// SIMATIC S7-200 project (STEP 7-Micro/WIN), CPU 224 REL 02.01

ORGANIZATION_BLOCK MAIN:OB1
TITLE=程序注释
BEGIN
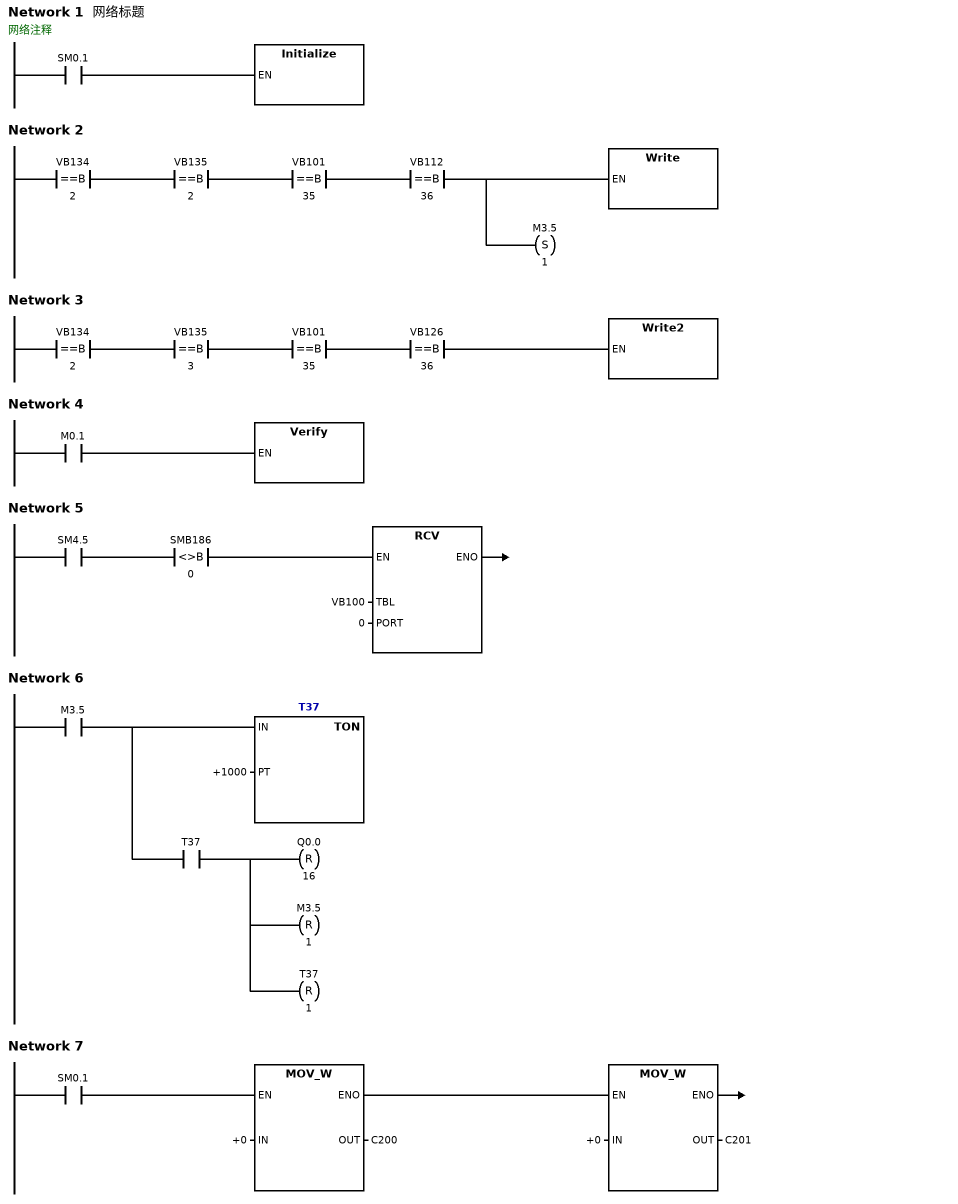
Network 1 // 网络标题
// 网络注释
LD     SM0.1
CALL   Initialize:SBR3
Network 2
LDB=   VB134, 2
AB=    VB135, 2
AB=    VB101, 35
AB=    VB112, 36
CALL   Write:SBR1
S      M3.5, 1
Network 3
LDB=   VB134, 2
AB=    VB135, 3
AB=    VB101, 35
AB=    VB126, 36
CALL   Write2:SBR6
Network 4
LD     M0.1
CALL   Verify:SBR2
Network 5
LD     SM4.5
AB<>   SMB186, 0
RCV    VB100, 0
Network 6
LD     M3.5
TON    T37, +1000
A      T37
R      Q0.0, 16
R      M3.5, 1
R      T37, 1
Network 7
LD     SM0.1
MOVW   +0, C200
AENO
MOVW   +0, C201
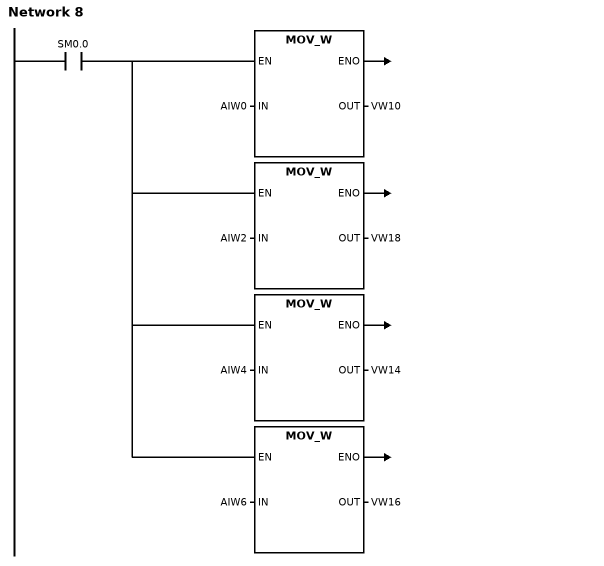
Network 8
LD     SM0.0
MOVW   AIW0, VW10
MOVW   AIW2, VW18
MOVW   AIW4, VW14
MOVW   AIW6, VW16
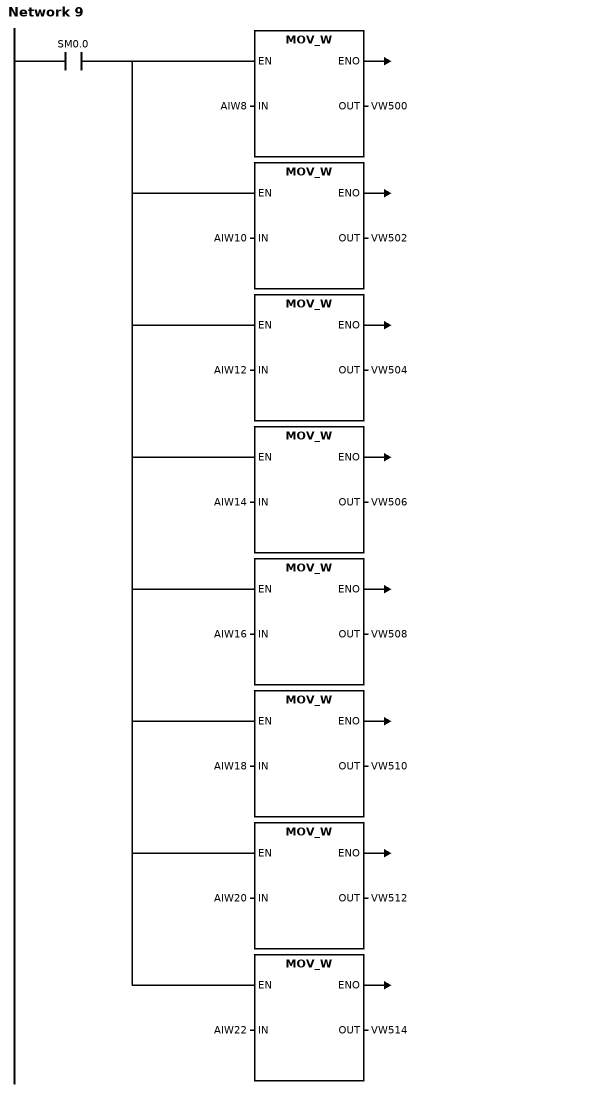
Network 9
LD     SM0.0
MOVW   AIW8, VW500
MOVW   AIW10, VW502
MOVW   AIW12, VW504
MOVW   AIW14, VW506
MOVW   AIW16, VW508
MOVW   AIW18, VW510
MOVW   AIW20, VW512
MOVW   AIW22, VW514
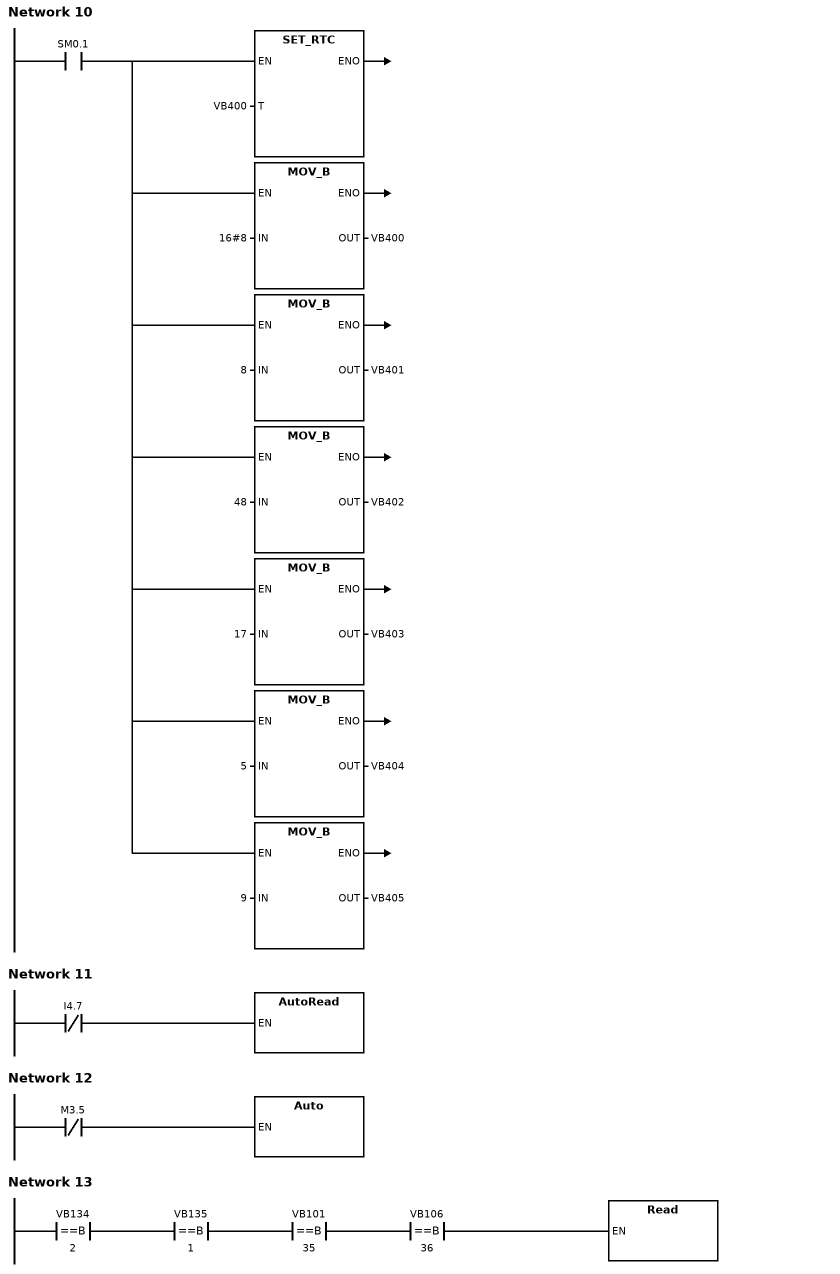
Network 10
LD     SM0.1
TODW   VB400
MOVB   16#8, VB400
MOVB   8, VB401
MOVB   48, VB402
MOVB   17, VB403
MOVB   5, VB404
MOVB   9, VB405
Network 11
LDN    I4.7
CALL   AutoRead:SBR5
Network 12
LDN    M3.5
CALL   Auto:SBR4
Network 13
LDB=   VB134, 2
AB=    VB135, 1
AB=    VB101, 35
AB=    VB106, 36
CALL   Read:SBR0
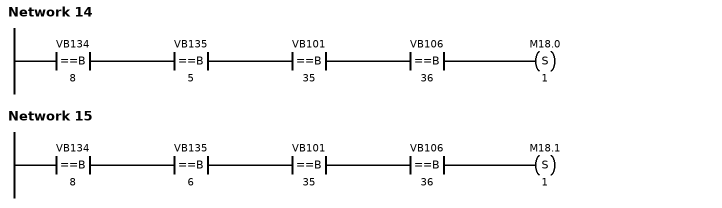
Network 14
LDB=   VB134, 8
AB=    VB135, 5
AB=    VB101, 35
AB=    VB106, 36
S      M18.0, 1
Network 15
LDB=   VB134, 8
AB=    VB135, 6
AB=    VB101, 35
AB=    VB106, 36
S      M18.1, 1
END_ORGANIZATION_BLOCK

SUBROUTINE_BLOCK Read:SBR0
TITLE=子程序注释
BEGIN
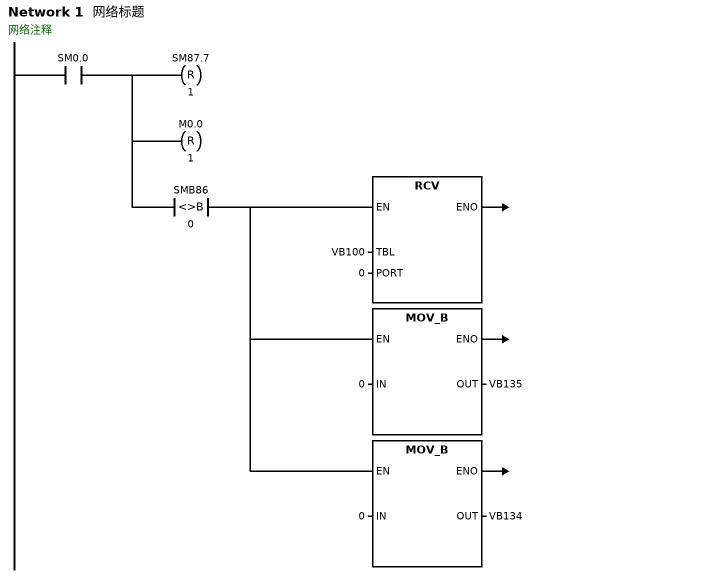
Network 1 // 网络标题
// 网络注释
LD     SM0.0
R      SM87.7, 1
R      M0.0, 1
AB<>   SMB86, 0
RCV    VB100, 0
MOVB   0, VB135
MOVB   0, VB134
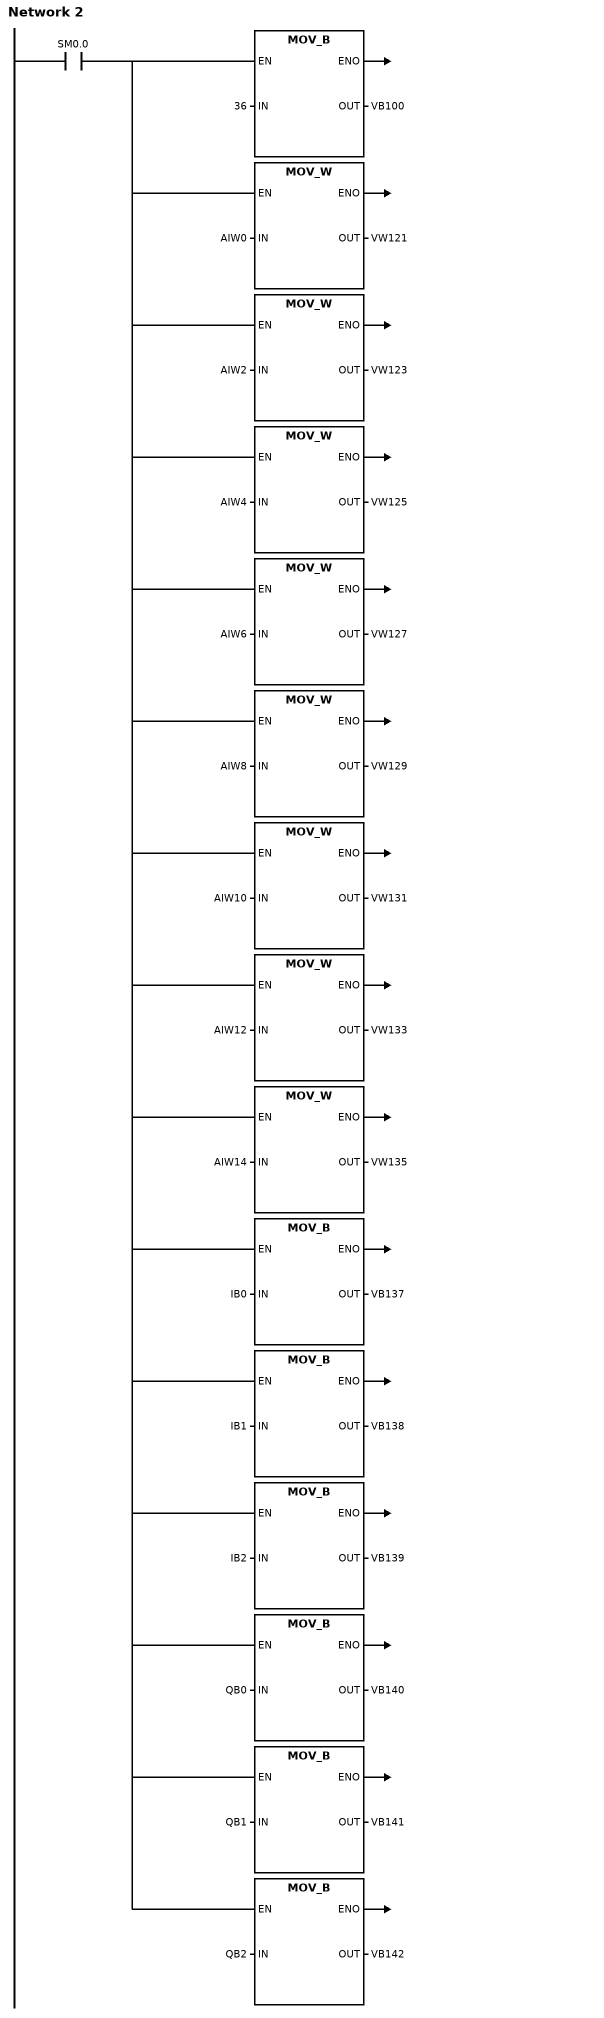
Network 2
LD     SM0.0
MOVB   36, VB100
MOVW   AIW0, VW121
MOVW   AIW2, VW123
MOVW   AIW4, VW125
MOVW   AIW6, VW127
MOVW   AIW8, VW129
MOVW   AIW10, VW131
MOVW   AIW12, VW133
MOVW   AIW14, VW135
MOVB   IB0, VB137
MOVB   IB1, VB138
MOVB   IB2, VB139
MOVB   QB0, VB140
MOVB   QB1, VB141
MOVB   QB2, VB142
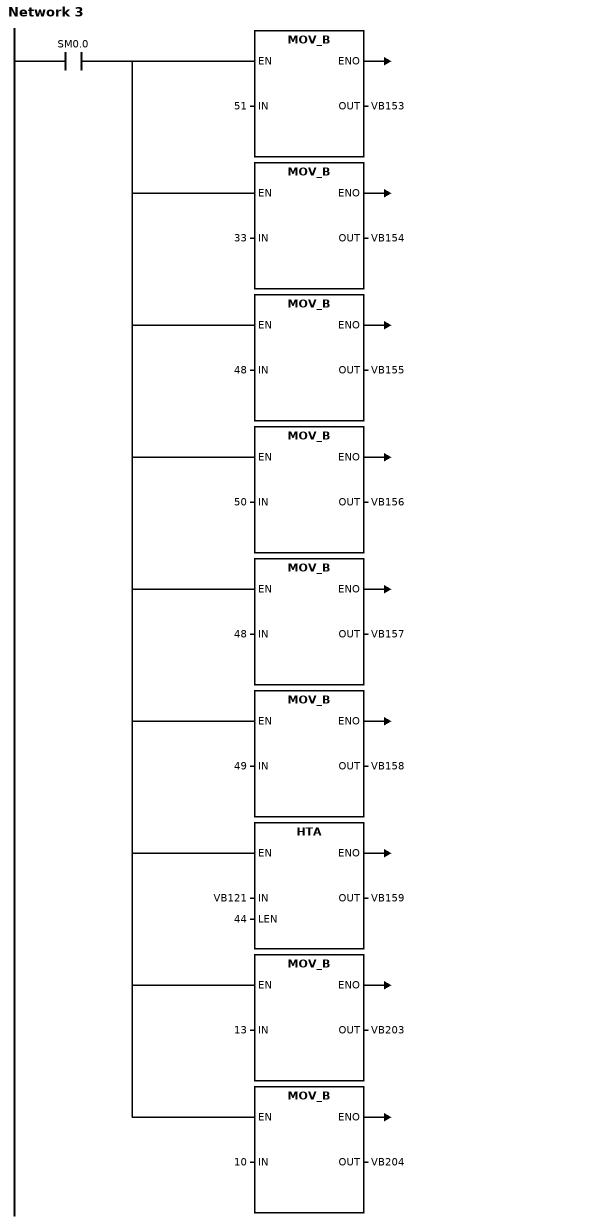
Network 3
LD     SM0.0
MOVB   51, VB153
MOVB   33, VB154
MOVB   48, VB155
MOVB   50, VB156
MOVB   48, VB157
MOVB   49, VB158
HTA    VB121, VB159, 44
MOVB   13, VB203
MOVB   10, VB204
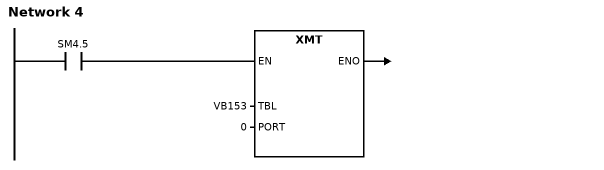
Network 4
LD     SM4.5
XMT    VB153, 0
END_SUBROUTINE_BLOCK

SUBROUTINE_BLOCK Write:SBR1
TITLE=
BEGIN
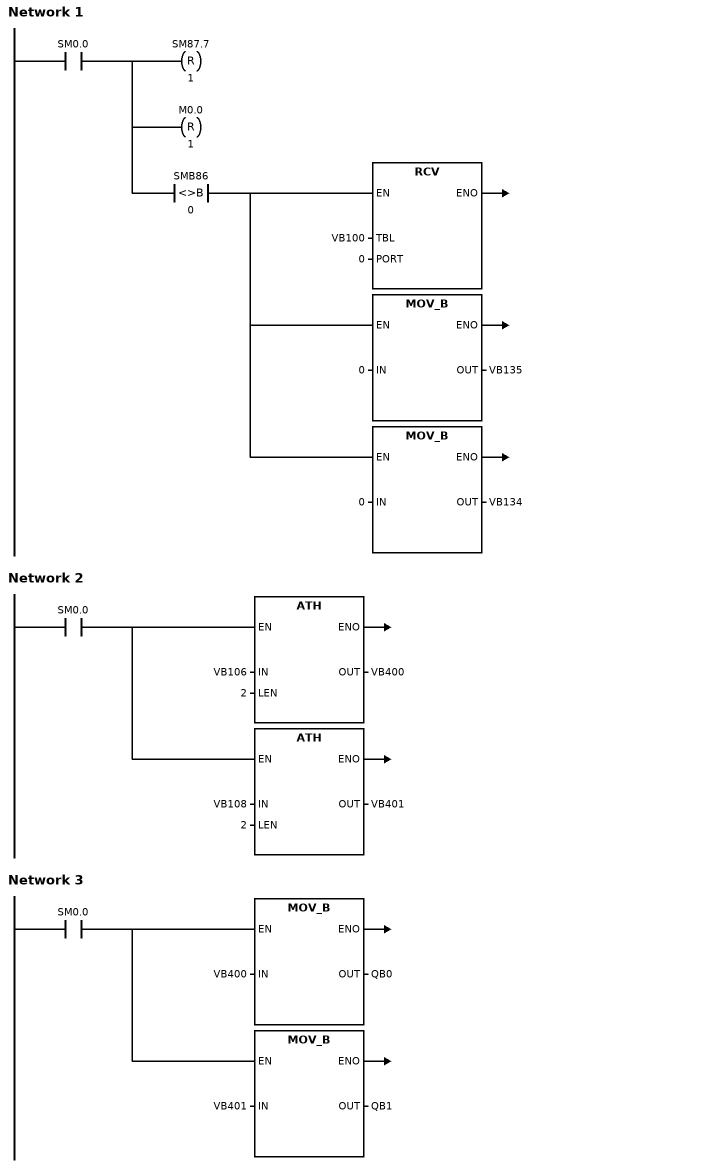
Network 1
LD     SM0.0
R      SM87.7, 1
R      M0.0, 1
AB<>   SMB86, 0
RCV    VB100, 0
MOVB   0, VB135
MOVB   0, VB134
Network 2
LD     SM0.0
ATH    VB106, VB400, 2
ATH    VB108, VB401, 2
Network 3
LD     SM0.0
MOVB   VB400, QB0
MOVB   VB401, QB1
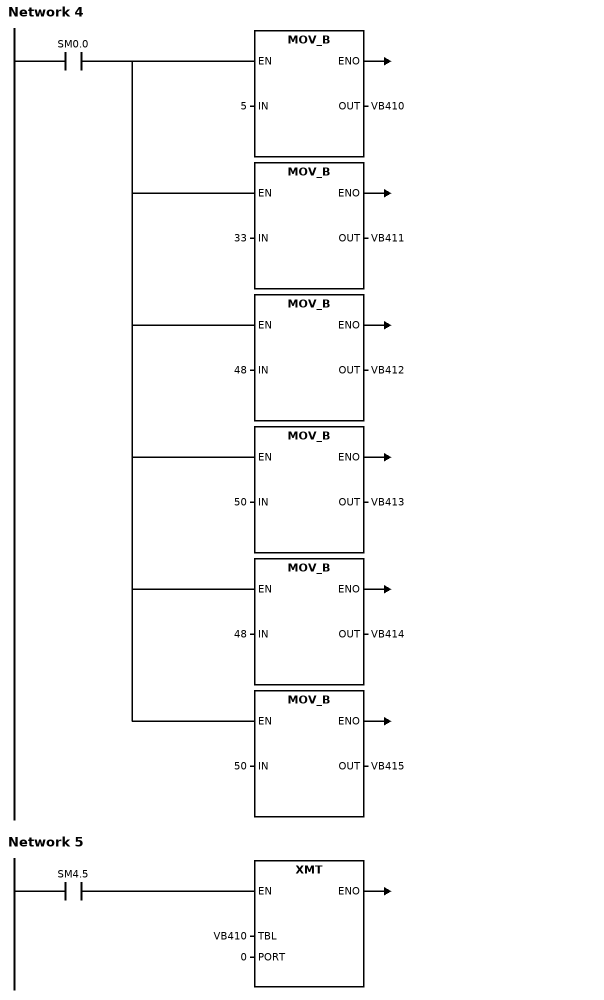
Network 4
LD     SM0.0
MOVB   5, VB410
MOVB   33, VB411
MOVB   48, VB412
MOVB   50, VB413
MOVB   48, VB414
MOVB   50, VB415
Network 5
LD     SM4.5
XMT    VB410, 0
END_SUBROUTINE_BLOCK

SUBROUTINE_BLOCK Verify:SBR2
TITLE=
BEGIN
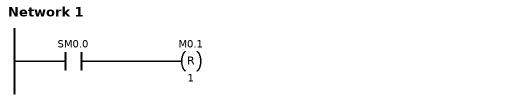
Network 1
LD     SM0.0
R      M0.1, 1
END_SUBROUTINE_BLOCK

SUBROUTINE_BLOCK Initialize:SBR3
TITLE=
BEGIN
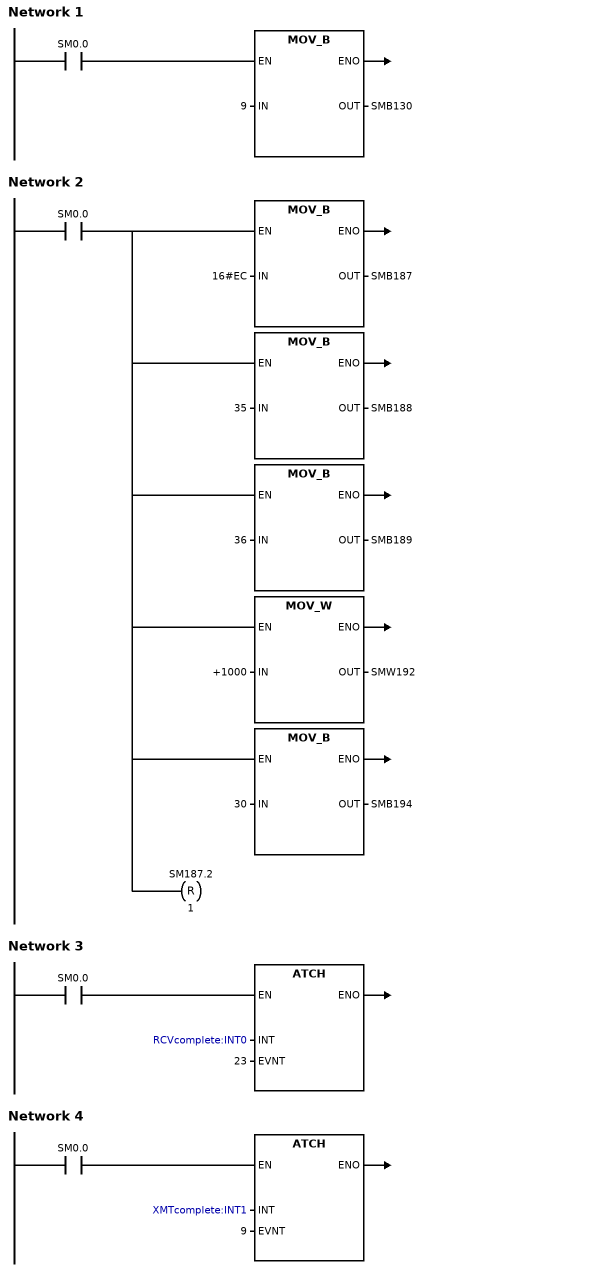
Network 1
LD     SM0.0
MOVB   9, SMB130
Network 2
LD     SM0.0
MOVB   16#EC, SMB187
MOVB   35, SMB188
MOVB   36, SMB189
MOVW   +1000, SMW192
MOVB   30, SMB194
R      SM187.2, 1
Network 3
LD     SM0.0
ATCH   RCVcomplete:INT0, 23
Network 4
LD     SM0.0
ATCH   XMTcomplete:INT1, 9
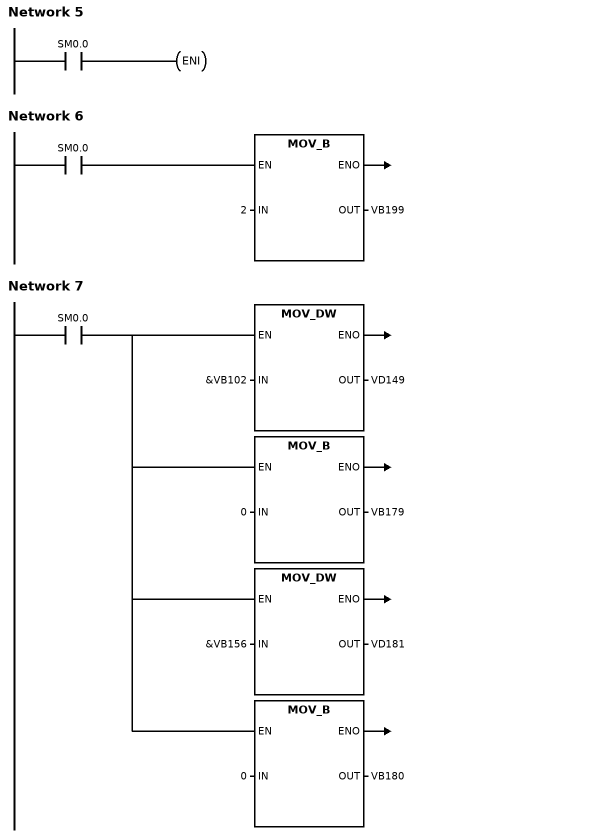
Network 5
LD     SM0.0
ENI
Network 6
LD     SM0.0
MOVB   2, VB199
Network 7
LD     SM0.0
MOVD   &VB102, VD149
MOVB   0, VB179
MOVD   &VB156, VD181
MOVB   0, VB180
END_SUBROUTINE_BLOCK

SUBROUTINE_BLOCK Auto:SBR4
TITLE=
BEGIN
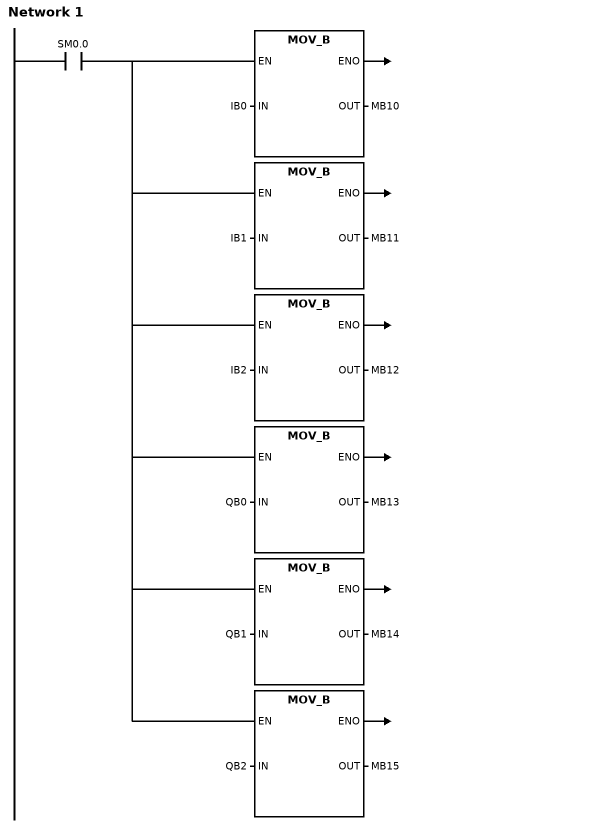
Network 1
LD     SM0.0
MOVB   IB0, MB10
MOVB   IB1, MB11
MOVB   IB2, MB12
MOVB   QB0, MB13
MOVB   QB1, MB14
MOVB   QB2, MB15
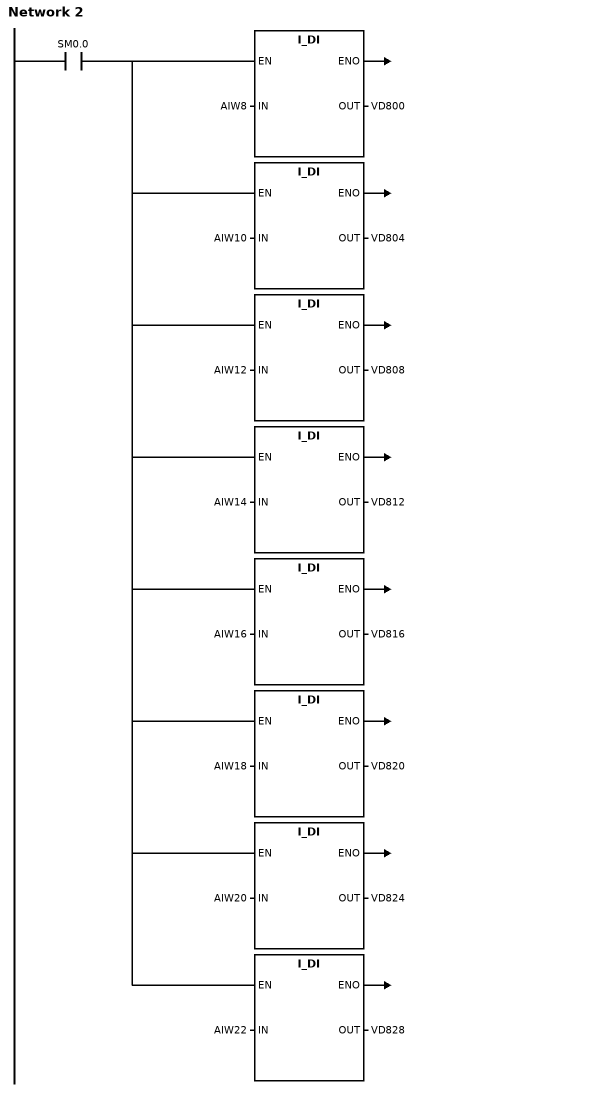
Network 2
LD     SM0.0
ITD    AIW8, VD800
ITD    AIW10, VD804
ITD    AIW12, VD808
ITD    AIW14, VD812
ITD    AIW16, VD816
ITD    AIW18, VD820
ITD    AIW20, VD824
ITD    AIW22, VD828
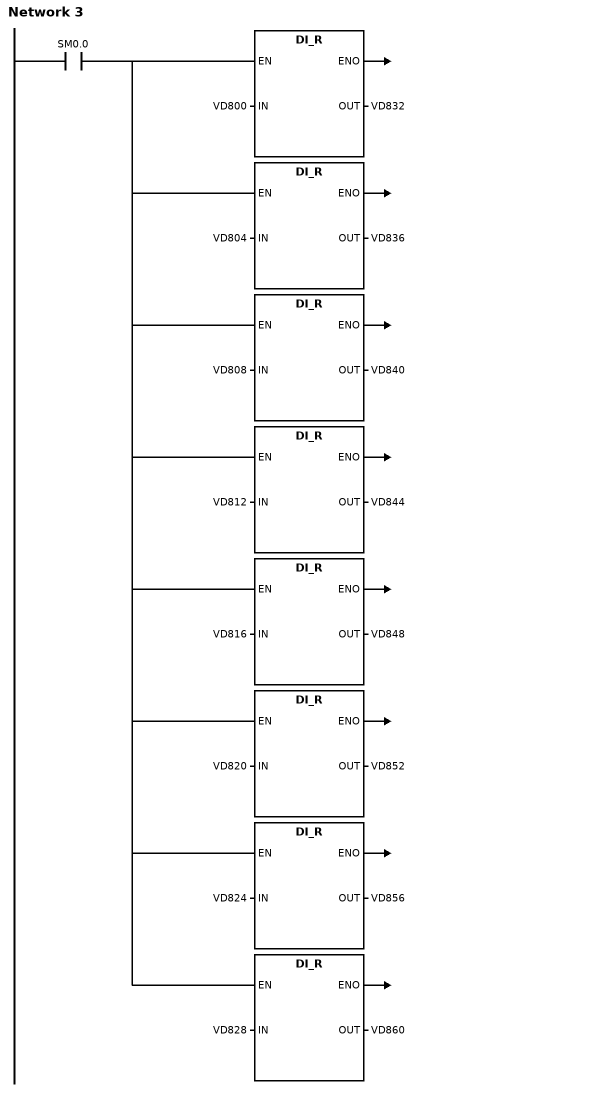
Network 3
LD     SM0.0
DTR    VD800, VD832
DTR    VD804, VD836
DTR    VD808, VD840
DTR    VD812, VD844
DTR    VD816, VD848
DTR    VD820, VD852
DTR    VD824, VD856
DTR    VD828, VD860
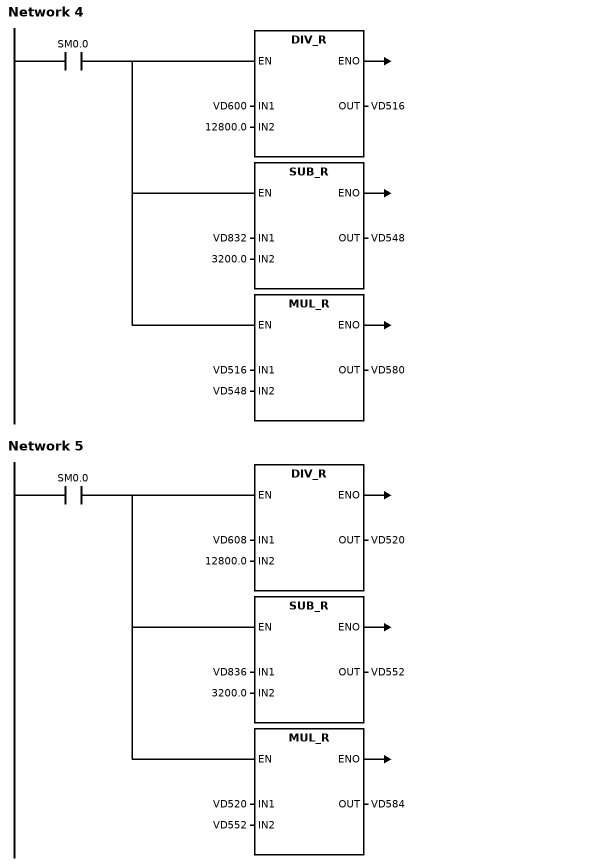
Network 4
LD     SM0.0
MOVR   VD600, VD516
/R     12800.0, VD516
MOVR   VD832, VD548
-R     3200.0, VD548
MOVR   VD516, VD580
*R     VD548, VD580
Network 5
LD     SM0.0
MOVR   VD608, VD520
/R     12800.0, VD520
MOVR   VD836, VD552
-R     3200.0, VD552
MOVR   VD520, VD584
*R     VD552, VD584
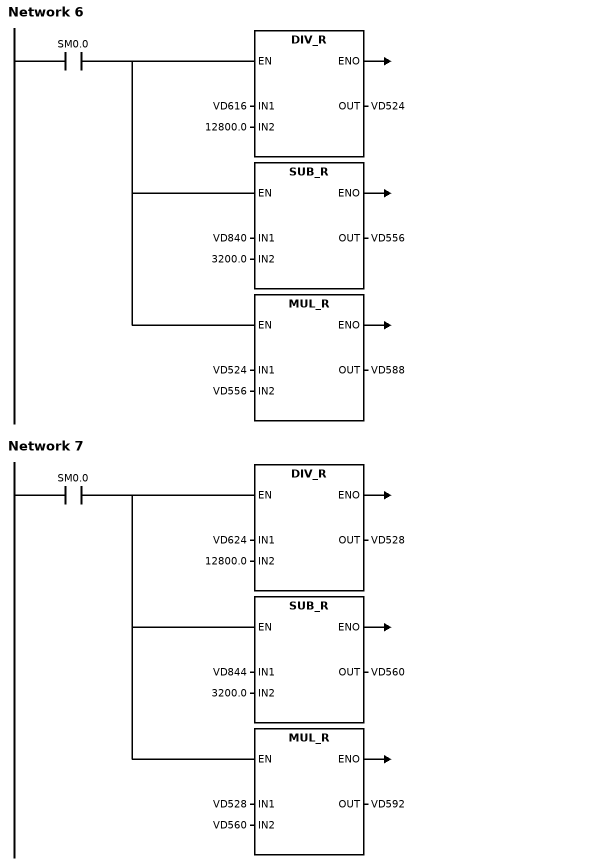
Network 6
LD     SM0.0
MOVR   VD616, VD524
/R     12800.0, VD524
MOVR   VD840, VD556
-R     3200.0, VD556
MOVR   VD524, VD588
*R     VD556, VD588
Network 7
LD     SM0.0
MOVR   VD624, VD528
/R     12800.0, VD528
MOVR   VD844, VD560
-R     3200.0, VD560
MOVR   VD528, VD592
*R     VD560, VD592
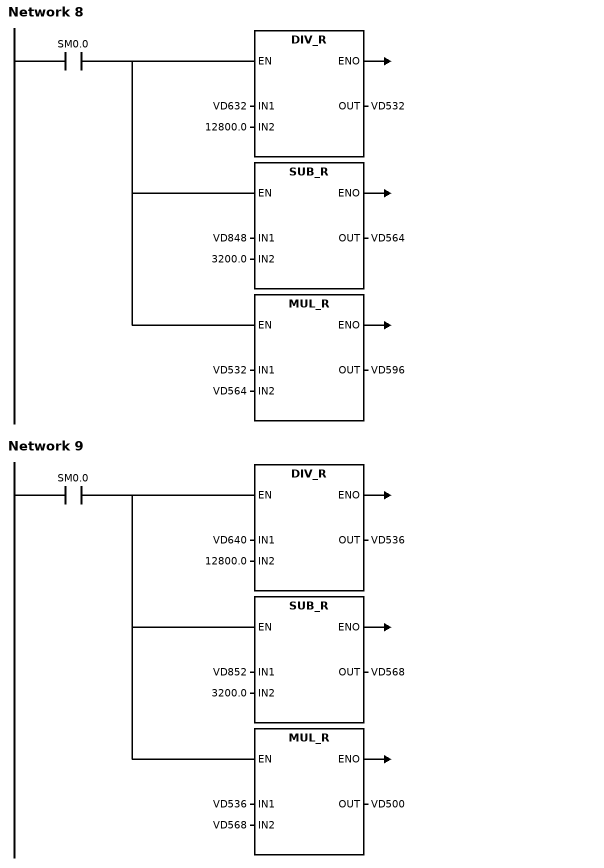
Network 8
LD     SM0.0
MOVR   VD632, VD532
/R     12800.0, VD532
MOVR   VD848, VD564
-R     3200.0, VD564
MOVR   VD532, VD596
*R     VD564, VD596
Network 9
LD     SM0.0
MOVR   VD640, VD536
/R     12800.0, VD536
MOVR   VD852, VD568
-R     3200.0, VD568
MOVR   VD536, VD500
*R     VD568, VD500
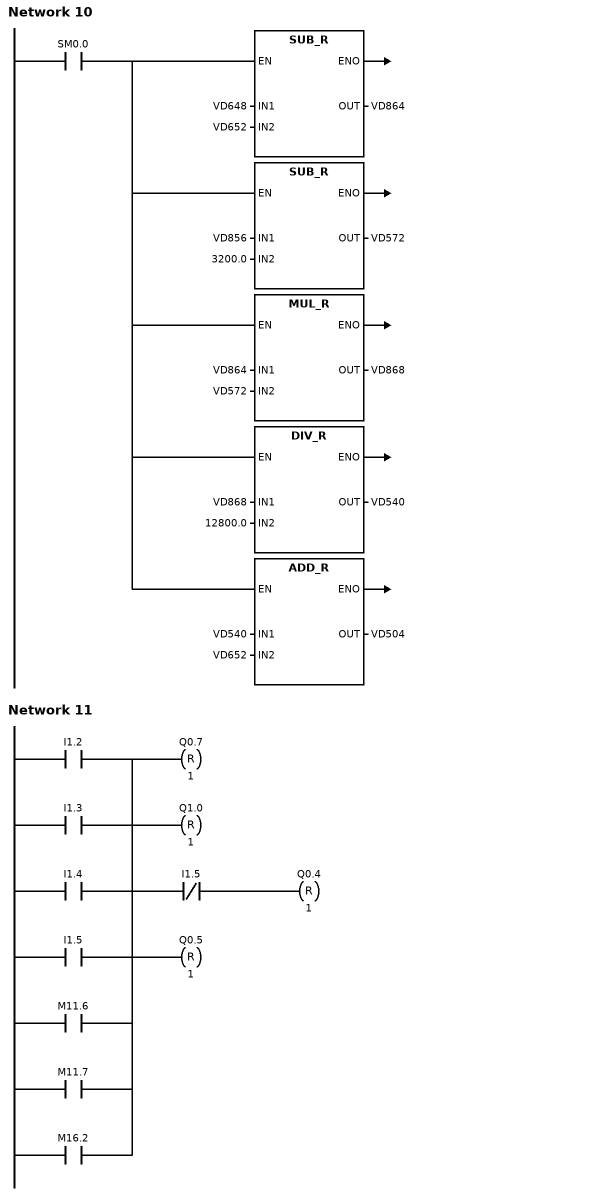
Network 10
LD     SM0.0
MOVR   VD648, VD864
-R     VD652, VD864
MOVR   VD856, VD572
-R     3200.0, VD572
MOVR   VD864, VD868
*R     VD572, VD868
MOVR   VD868, VD540
/R     12800.0, VD540
MOVR   VD540, VD504
+R     VD652, VD504
Network 11
LD     I1.2
O      I1.3
O      I1.4
O      I1.5
O      M11.6
O      M11.7
O      M16.2
LPS
R      Q0.7, 1
R      Q1.0, 1
AN     I1.5
R      Q0.4, 1
LPP
R      Q0.5, 1
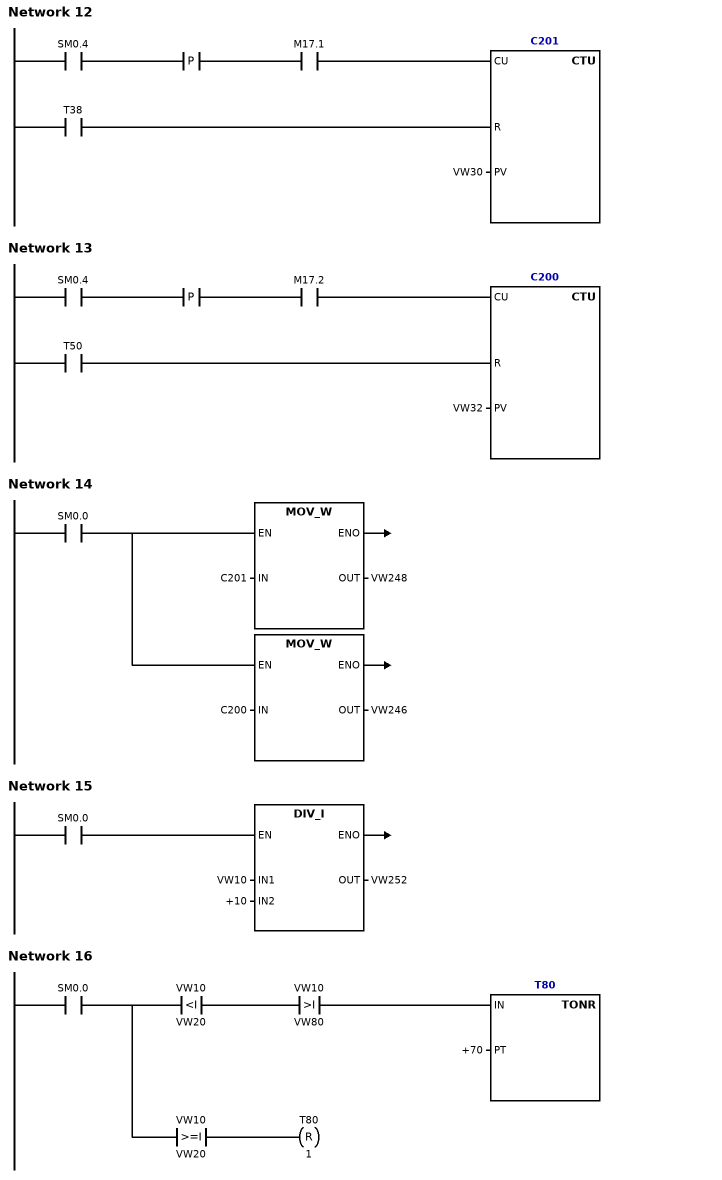
Network 12
LD     SM0.4
EU
A      M17.1
LD     T38
CTU    C201, VW30
Network 13
LD     SM0.4
EU
A      M17.2
LD     T50
CTU    C200, VW32
Network 14
LD     SM0.0
MOVW   C201, VW248
MOVW   C200, VW246
Network 15
LD     SM0.0
MOVW   VW10, VW252
/I     +10, VW252
Network 16
LD     SM0.0
LPS
AW<    VW10, VW20
AW>    VW10, VW80
TONR   T80, +70
LPP
AW>=   VW10, VW20
R      T80, 1
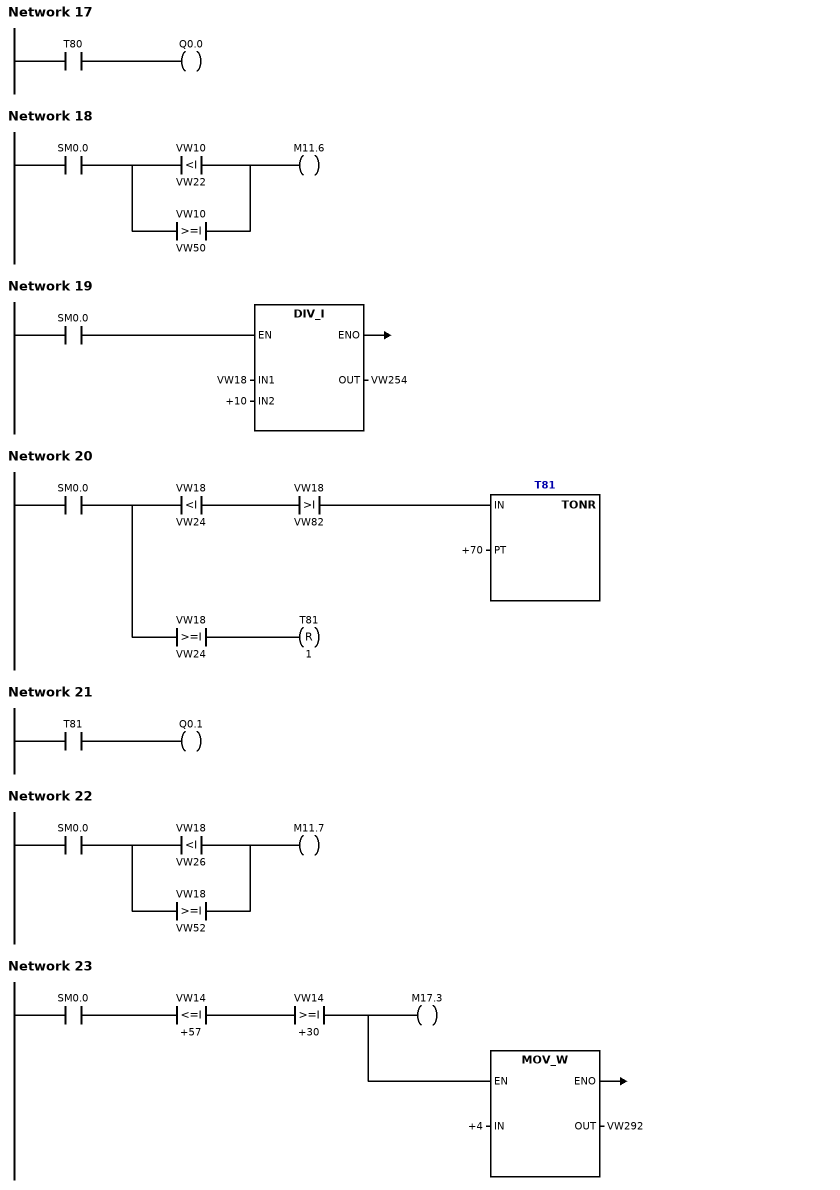
Network 17
LD     T80
=      Q0.0
Network 18
LD     SM0.0
LDW<   VW10, VW22
OW>=   VW10, VW50
ALD
=      M11.6
Network 19
LD     SM0.0
MOVW   VW18, VW254
/I     +10, VW254
Network 20
LD     SM0.0
LPS
AW<    VW18, VW24
AW>    VW18, VW82
TONR   T81, +70
LPP
AW>=   VW18, VW24
R      T81, 1
Network 21
LD     T81
=      Q0.1
Network 22
LD     SM0.0
LDW<   VW18, VW26
OW>=   VW18, VW52
ALD
=      M11.7
Network 23
LD     SM0.0
AW<=   VW14, +57
AW>=   VW14, +30
=      M17.3
MOVW   +4, VW292
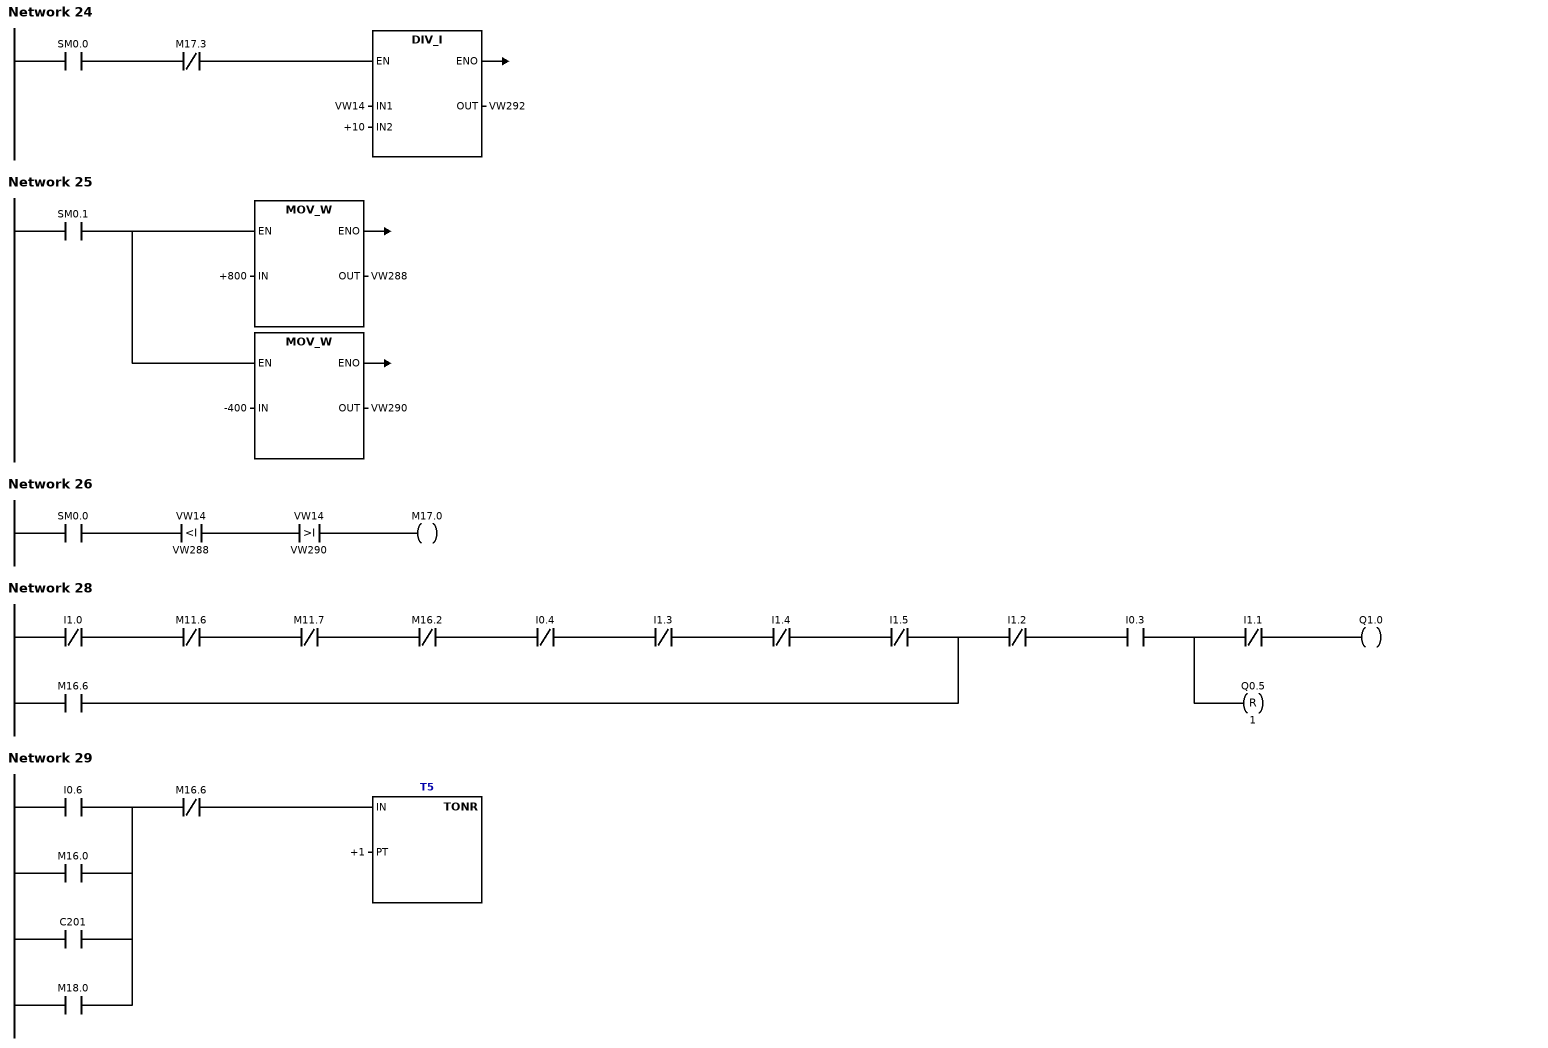
Network 24
LD     SM0.0
AN     M17.3
MOVW   VW14, VW292
/I     +10, VW292
Network 25
LD     SM0.1
MOVW   +800, VW288
MOVW   -400, VW290
Network 26
LD     SM0.0
AW<    VW14, VW288
AW>    VW14, VW290
=      M17.0
Network 28
LDN    I1.0
AN     M11.6
AN     M11.7
AN     M16.2
AN     I0.4
AN     I1.3
AN     I1.4
AN     I1.5
O      M16.6
AN     I1.2
A      I0.3
LPS
AN     I1.1
=      Q1.0
LPP
R      Q0.5, 1
Network 29
LD     I0.6
O      M16.0
O      C201
O      M18.0
AN     M16.6
TONR   T5, +1
